Universal Robots PolyScope program: d_up.urp

Program d_up (installation=string_planes directory=/programs createdIn=5.17.3 lastSavedIn=5.17.3 robotSerialNumber=20245501435)
Calibrated DH parameters: a=[0.000154, -0.137004, -0.385524, -0.00002, 0.000092, 0]; d=[0.162441, 211.794786, -230.585024, 18.923638, 0.099786, 0.09951]; alpha=[1.569493, -0.001902, 0.003874, 1.570111, -1.570167, 0]; deltaTheta=[0, -1.242934, 1.056292, 0.186646, 0.000002, 0.000001]
InitVariablesNode
Robot Program (runOnlyOnce=false)
  MoveL speed 250 mm/s, acceleration 1200 mm/s^2 (useActiveTCP=true) feature=Plane_2
    Waypoint Waypoint_3: TCP in base x=384.493 y=289.417 z=153.372 mm, rx=-1.5873 ry=-2.1561 rz=1.2208 rad; joints [-163.891, -53.511, 112.643, -101.372, -107.942, -172.933] deg; TCP offset x=28.21 y=-96.107 z=-99.69 mm, rx=0 ry=0 rz=0 rad; feature pose in base x=343.605 y=747.803 z=100.778 mm, rx=2.7685 ry=0.1285 rz=1.3673 rad
    Waypoint Waypoint_1: TCP in base x=331.971 y=722.315 z=108.291 mm, rx=-1.645 ry=-2.1081 rz=1.0591 rad; joints [-129.709, -21.469, 51.981, -76.268, -76.862, -148.975] deg; feature pose in base x=343.605 y=747.803 z=100.778 mm, rx=2.7685 ry=0.1285 rz=1.3673 rad
